// TIA Portal V18 export
VAR_GLOBAL   // PLC tag table "System Variables"
   RotaryCounts AT %MD100 : DInt;   // Actually rotary count feedback
   RotaryRPM AT %MD104 : Real;   // frequency of rotray feedack
   AuxPumpRunning AT %M10.0 : Bool;   // Status of Aux Pump. 1 Running 0 stopped
   EngineRPMCounts AT %MD108 : DInt;   // CAT Engine RPM count return
   EngineRPMFreq AT %MD112 : Real;   // CAT Engine RPM freqency measured
   CoolingFanRunning AT %M10.1 : Bool;   // Status of Cooler Running 0 stopped
   M1Running AT %M10.2 : Bool;   // Status of P1 Running 0 stopped
   M2Running AT %M10.3 : Bool;   // Status of P2 Running 0 stopped
   AuxPumpHOA AT %M10.4 : Bool;   // Actual Signal to Soft Starter
   CoolingFanHOA AT %M10.5 : Bool;   // Actual Signal to Soft Starter
   M1HOA AT %M10.6 : Bool;   // Actual Signal to Soft Starter
   M2HOA AT %M10.7 : Bool;   // Actual Signal to Soft Starter
   ChargePump1PSw AT %M11.0 : Bool;   // Close = Pressure
   TDLubeFlowSw AT %M11.1 : Bool;   // Close = Flow
   TankLowLevelSw AT %M11.2 : Bool;   // Low Level = Open
   TankHighTempSw AT %M11.3 : Bool;   // High Temp = Open
   TDFwdFilter2 AT %M11.5 : Bool;   // Plugged = Open
   TDRevFilter1 AT %M11.6 : Bool;   // Plugged = Open
   TDRevFilter2 AT %M11.7 : Bool;   // Plugged = Open
   AuxReturnFilter AT %M12.0 : Bool;   // Plugged = Open
   KLoopFilter AT %M12.1 : Bool;   // Plugged = Open
   ChargeFilter AT %M12.2 : Bool;   // Plugged = Open
   M1CurrentRaw AT %MW122 : Int;
   M2CurrentRaw AT %MW128 : Int;
   M1CurrentV AT %MD124 : Real;
   M2CurrentV AT %MD130 : Real;
   TDPressFWDRaw AT %MW134 : Int;   // TD Forward Pressure Input
   TDPressREVRaw AT %MW136 : Int;   // TD Reverse Pressure Input
   ClosedLoopTempRaw AT %MW138 : Int;
   ChargeFlowRaw AT %MW140 : Int;
   HotOilShuttleFlowRaw AT %MW142 : Int;
   AuxFlowRaw AT %MW144 : Int;
   ChargePress1Raw AT %MW146 : Int;
   ChargePress2Raw AT %MW148 : Int;
   TDPressFWDmA AT %MD150 : Real;   // TD Forward Pressure Input
   TDPressREVmA AT %MD154 : Real;   // TD Reverse Pressure Input
   ClosedLoopTempmA AT %MD158 : Real;
   ChargeFlowmA AT %MD162 : Real;
   HotOilShuttleFlowmA AT %MD166 : Real;
   AuxFlowmA AT %MD170 : Real;
   ChargePress1mA AT %MD174 : Real;
   ChargePress2mA AT %MD178 : Real;
   TDP1FwdCmdActRaw AT %MW182 : Int;   // Actual measured output to valve from module
   TDP1RevCmdActRaw AT %MW184 : Int;   // Actual measured output to valve from module
   TDP2FwdCmdActRaw AT %MW186 : Int;   // Actual measured output to valve from module
   TDP2RevCmdActRaw AT %MW188 : Int;   // Actual measured output to valve from module
   TDTorqCmdActRaw AT %MW190 : Int;   // Raw Output to card
   TDP1FwdCmdActmA AT %MD192 : Real;   // Actual measured output to valve from module
   TDP1RevCmdActmA AT %MD196 : Real;   // Actual measured output to valve from module
   TDP2FwdCmdActmA AT %MD200 : Real;   // Actual measured output to valve from module
   TDP2RevCmdActmA AT %MD204 : Real;   // Actual measured output to valve from module
   TDTorqCmdActmA AT %MD208 : Real;   // Actual measured output to valve from module
   LinkRetSw AT %M12.4 : Bool;   // Console Input
   TDAuxSw AT %M12.5 : Bool;   // Console Input
   LinkExtSw AT %M12.6 : Bool;   // Console Input
   TDEnSW AT %M12.7 : Bool;   // Console Input
   HSLT_Sw AT %M13.0 : Bool;   // Console Input
   HandlerFwdSw AT %M13.1 : Bool;   // Console Input
   HandlerRevSw AT %M13.2 : Bool;   // Console Input
   MPNotRunning AT %M13.3 : Bool;   // 0 Pump Running, 1 Pump Not Running - Allowed to Run. Power to permit
   QuillLockSw AT %M13.4 : Bool;   // Console Input
   BUWClSw AT %M13.5 : Bool;   // Console Input
   BUWDnSw AT %M13.6 : Bool;   // Console Input
   BUWUpSw AT %M13.7 : Bool;   // Console Input
   TDModeMUSpinSw AT %M14.0 : Bool;   // Console Input
   TDModeMUTorqSw AT %M14.1 : Bool;   // Console Input
   TDModeDrillRevSw AT %M14.2 : Bool;   // Console Input
   TDModeBreakOutSw AT %M14.3 : Bool;   // Console Input
   ElevOpSw AT %M14.4 : Bool;   // Console Input
   TDExtSw AT %M14.5 : Bool;   // Console Input
   ElevClSw AT %M14.6 : Bool;   // Console Input
   TDRetSw AT %M14.7 : Bool;   // Console Input
   PTO_Sw AT %M15.0 : Bool;   // Console Input
   PurgePressureSw AT %M15.1 : Bool;   // Console Input
   MSVClSw AT %M15.2 : Bool;   // Console Input
   MSVAutoSw AT %M15.3 : Bool;   // Console Input
   MSVOpSw AT %M15.4 : Bool;   // Console Input
   LinkFloatSw AT %M15.5 : Bool;   // Console Input
   MUTorqPotRaw AT %MW212 : Int;
   DrillTorqPotRaw AT %MW214 : Int;
   DrillThrottlePotRaw AT %MW216 : Int;
   MUTorqPotV AT %MD218 : Real;
   DrillTorqPotV AT %MD222 : Real;
   DrillThrottlePotV AT %MD226 : Real;
   RotEncLDSlot AT %MB230 : Byte;   // Bit 0-3 Slot 0, Bit 4-7 Slot 1. 0 0 0 0 for Idle, 0 0 0 1 Load Counter
   TDFwdPress1Raw AT %MD240 : UDInt;   // Pump 1 Forward Pressure output
   TDFwdPress2Raw AT %MD244 : UDInt;   // Pump 2 Forward Pressure output
   TDRevPress1Raw AT %MD248 : UDInt;   // Pump 1 Rev Pressure output
   TDRevPress2Raw AT %MD252 : UDInt;   // Pump 2 Rev Pressure output
   TDTorqPressRaw AT %MD256 : UDInt;   // Torq Output
   TDFwdPress1En AT %M15.6 : Bool;   // Enable Pump 1 Forward Pressure output
   TDFwdPress2En AT %M15.7 : Bool;   // Enable Pump 2 Forward Pressure output
   TDRevPress1En AT %M16.0 : Bool;   // Enable Pump 1 Rev Pressure output
   TDRevPress2En AT %M16.1 : Bool;   // Enable Pump 2 Rev Pressure output
   TDTorqPressEn AT %M16.2 : Bool;   // Enable Torq output
   BUWClSol AT %M16.4 : Bool;
   HSLT_Sol AT %M16.5 : Bool;
   ElevClSol AT %M16.6 : Bool;
   ElevOpSol AT %M16.7 : Bool;
   LinkExtSol AT %M17.0 : Bool;
   LinkRetSol AT %M17.1 : Bool;
   LinkFloatSol AT %M17.2 : Bool;
   LSHT_Sol AT %M17.3 : Bool;
   MSVOpSol AT %M17.4 : Bool;
   MSVClSol AT %M17.5 : Bool;
   BUWDnSol AT %M17.6 : Bool;
   BUWUpSol AT %M17.7 : Bool;
   HandlerFWDSol AT %M18.0 : Bool;
   HandlerREVSol AT %M18.1 : Bool;
   TDExtSol AT %M18.2 : Bool;
   TDRetSol AT %M18.3 : Bool;   // Output Coil
   HourMeterOn AT %M18.4 : Bool;
   EngRampSpeedDn AT %M18.5 : Bool;
   AuxPumpStart AT %M18.6 : Bool;
   EngRampSpeedUp AT %M18.7 : Bool;
   CoolingFanStart AT %M19.0 : Bool;
   FailSafeEnSol AT %M19.1 : Bool;
   PumpEnSol AT %M19.2 : Bool;   // CAT/Rig 11 Only
   BOControlSol AT %M19.3 : Bool;
   AuxUnloaderSol AT %M19.4 : Bool;
   HotOilControlSol AT %M19.5 : Bool;
   BUWOpSol AT %M19.6 : Bool;
   BypassValveSol AT %M19.7 : Bool;
   TDFwdPress1mA AT %MD260 : Real;   // Pump 1 Forward Pressure output
   TDFwdPress2mA AT %MD264 : Real;   // Pump 2 Forward Pressure output
   TDRevPress1mA AT %MD268 : Real;   // Pump 1 Rev Pressure output
   TDRevPress2mA AT %MD272 : Real;   // Pump 2 Rev Pressure output
   TDTorqPressmA AT %MD276 : Real;   // Torq Output
   PTOLED AT %M20.4 : Bool;
   HPUFaultLED AT %M20.5 : Bool;
   TDFlushFaultLED AT %M20.6 : Bool;
   BUWClLED AT %M20.7 : Bool;
   TDEnLED AT %M21.0 : Bool;
   ConLowPurgeLED AT %M21.1 : Bool;
   MSVClLED AT %M21.2 : Bool;   // Mud Saver valve closed LED
   QuillLockLED AT %M21.3 : Bool;
   ElevClLED AT %M21.4 : Bool;
   Horn AT %M21.5 : Bool;
   MSVClInt AT %M21.6 : Bool;   // Mud saver valve closed interlocks outputs
   BUWClInt AT %M21.7 : Bool;   // BUW Closed interlock outputs
   DrillRecTorqRaw AT %MW280 : Int;
   DrillRecRPMRaw AT %MW282 : Int;
   DrillRecTorqFtLbs AT %MD284 : Real;
   DrillRecRPM AT %MD288 : Real;
   DrillRecTorqmA AT %MD292 : Real;
   DrillRecRPMmA AT %MD296 : Real;
   RotEncUnFl AT %M22.0 : Bool;   // Encoder underflow
   RotEncOvFl AT %M22.1 : Bool;   // Encoder OVerflow
   RotEncPosReset AT %M22.2 : Bool;   // Set high to trigger zero position of encoder. Bit will reset once position reset
   RotEncSlot0 AT %MD232 : Real;
   RotEncSlot1 AT %MD236 : Real;
   TDRotStopped AT %M22.3 : Bool;   // Set if TD has not moved after stop time elapsed
   RotAbsPosDeg AT %MD300 : Real;   // Absolute rotary position from zero point
   RotRelPosDeg AT %MD304 : Real;   // Position from 0-360 degrees
   RotPosTurns AT %MD308 : Real;   // Turns from zero point
   TDFlushFlowSw AT %M22.4 : Bool;
   M1Current AT %MD312 : Real;
   M2Current AT %MD316 : Real;
   TDPressFwdPSI AT %MD320 : Real;   // TD Fwd Pressure PSI
   TDPressRevPSI AT %MD324 : Real;   // TD Rev Pressure PSI
   ClosedLoopTempC AT %MD328 : Real;   // Closed Loop Temp in C
   ChargeFlowGPM AT %MD332 : Real;   // Charge Flow in GPM
   HotOilFlowGPM AT %MD336 : Real;   // Hot Oil Shuttle Flow in GPM
   AuxFlowGPM AT %MD340 : Real;   // Aux Flow GPM
   ChargePress1PSI AT %MD344 : Real;   // Charge Pump 1 Pressure PSI
   ChargePress2PSI AT %MD348 : Real;   // Charge Pump 2 Pressure PSI
   M1CurrentFilt AT %MD352 : Real;
   M2CurrentFilt AT %MD356 : Real;
   TDPressFwdPSIFilt AT %MD360 : Real;
   TDPressRevPSIFilt AT %MD364 : Real;
   ClosedLoopTempCFilt AT %MD368 : Real;
   ChargeFlowGPMFilt AT %MD372 : Real;
   HotOilFlowGPMFilt AT %MD376 : Real;
   AuxFlowGPMFilt AT %MD380 : Real;
   ChargePress1PSIFilt AT %MD384 : Real;
   ChargePress2PSIFilt AT %MD388 : Real;
   AuxPumpHand AT %M22.5 : Bool;   // Starter HOA switch in the Hand Position
   AuxPumpOff AT %M22.6 : Bool;   // Starter HOA switch in the Off position
   CoolingFanHand AT %M23.0 : Bool;   // Starter HOA switch in the Hand Position
   CoolingFanOff AT %M23.1 : Bool;   // Starter HOA switch in the Off position
   M1Hand AT %M23.3 : Bool;   // Starter HOA switch in the Hand Position
   M1Off AT %M23.4 : Bool;   // Starter HOA switch in the Off position
   M2Hand AT %M23.6 : Bool;   // Starter HOA switch in the Hand Position
   M2Off AT %M23.7 : Bool;   // Starter HOA switch in the Off position
   AuxPumpFault AT %M22.7 : Bool;   // Motor failed to start before motor timeout time
   CoolingFanFault AT %M23.2 : Bool;   // Motor failed to start before motor timeout time
   M1Fault AT %M23.5 : Bool;   // Motor failed to start before motor timeout time
   M2Fault AT %M24.0 : Bool;   // Motor failed to start before motor timeout time
   M1Start AT %M20.2 : Bool;   // Start Motor 1
   M2Start AT %M20.3 : Bool;   // Start Motor 2
   BypassStart AT %M24.1 : Bool;   // Ready for Bypass to start, waiting for PTO
   BypassRunning AT %M24.2 : Bool;   // Latched Signal set if PTO pressed after Bypass Start
   StartCAT AT %M24.3 : Bool;   // Indicates CAT startup up. System ramps up and will enable.
   BUWMaintConfirm AT %M24.4 : Bool;
   PTOConfirmed AT %M24.5 : Bool;   // PTO Confirm pulse for 5 seconds after button pressed
   BUWOpenClk AT %M24.6 : Bool;   // Periodic clock signal that will be on for 5 seconds and off for 1 min. Used for maintain gripper open
   BUWAutoCl AT %M24.7 : Bool;   // Latch for Gripper Close
   BUWAutoClHold AT %M25.0 : Bool;   // LAtch for Gripper Hold Closed
   BUWAutoOp AT %M25.1 : Bool;   // Lath for Gripper Open
   OscSpeedfwdHold AT %M25.2 : Bool;
   QuillLockEnabled AT %M25.3 : Bool;   // Bit used to know if Quill Lock allowed
   BUWClHoldTime AT %M25.4 : Bool;   // On for half a second to hold the close before turning off
   MUTorqPotPer AT %MD392 : Real;
   DrillTorqPotPer AT %MD396 : Real;
   DrillThrottlePotPer AT %MD400 : Real;
   MUTorqPotPerFilt AT %MD404 : Real;
   DrillTorqPotPerFilt AT %MD408 : Real;
   DrillThrottlePotPerFilt AT %MD412 : Real;
   ActTorqFtLbs AT %MD416 : Real;   // Calculated actual torque
   ActTorqFtLbsFilt AT %MD420 : Real;   // Filtered Actual Torque
   TDDifPressPSI AT %MD424 : Real;   // Diffential pressure betweeen FWD and REV
   DrillTorqSetFtLbs AT %MD428 : Real;   // Internal setpoint value from the console input FtLbs
   MUTorqSetFtLbs AT %MD432 : Real;   // Internal setpoint value from the console input FtLbs
   RotDegPerCount AT %MD436 : Real;   // Actual Degrees per Count for current encoder setup
   DrillTorqSetMax AT %MD440 : Real;   // Maximum value allowed to set drill torq too based on MU torq settings
   BOCycleDone AT %M25.6 : Bool;   // Trigger when BO Sw released
   MUCycleDone AT %M25.7 : Bool;   // Set when MU done
   MUSwRelease AT %M26.0 : Bool;   // Trigger when MU SW released
   MUDoneSetFtLbs AT %MD444 : Real;   // Minimum torque to surpass to declare MU Done
   ElevClFeedback AT %M12.3 : Bool;   // Feedback switch that the elevators are closed
   LamptTest AT %M26.1 : Bool;   // Bit Used to trigger Lamp to turn on.
   FlushFaultNoSpin AT %M26.2 : Bool;   // TD flush faulted. No Spin allowed
   ThrottleDisable AT %M26.3 : Bool;   // Throttle disable if high
   ThrottleUnlocked AT %M26.4 : Bool;   // Throttle boots up locked. Must be below zero to enable after startup
   DrillTorqLimited AT %M26.5 : Bool;   // Set high if max drill torq limited by max makeup torq
   DrillTorqSetPSI AT %MD448 : Real;   // PSI equivalent to get desired torq from valve
   MUTorqSetPSI AT %MD452 : Real;   // PSI equivalent to get desired torq from valve
   TDStart AT %M25.5 : Bool;   // Bit will be set High when TD is started for regular operations
   BypassPTO AT %M26.6 : Bool;   // Bypass PTO accept
   BypassOutEnable AT %M26.7 : Bool;   // Bypass control enabled to allow signal to Pumps after delay
   BypassHighTemp AT %M27.0 : Bool;   // High Closed loop temp in bypass mode
   TDPressTxFault AT %M27.1 : Bool;   // One of the pressure transducers if not working. No auto MU
   HSLTDisThrottle AT %M27.2 : Bool;   // Bit high after shift to disable throttle
   LSHTDisThrottle AT %M27.3 : Bool;   // Bit high after shift to disable throttle
   MUSeqRunning AT %M27.4 : Bool;   // Bool indicating mak up sequence is running.
   AutoMUTorqLow AT %M27.5 : Bool;   // Auto Make Up Low Torque range
   AutoMUTorqMid AT %M27.6 : Bool;   // Auto Make Up Mid Torque Range
   AutoMuTorqHigh AT %M27.7 : Bool;   // Auto Make Up High Torque Range
   HiTempRPMRed AT %M28.1 : Bool;   // Bit indicating high temperature and RPM to be reduced
   HiTempShutdown AT %M28.2 : Bool;   // Bit indicating high temperature and shutdown needed.
   TDRotDirFwd AT %M28.3 : Bool;   // Rotary moving fwd
   TDRotDirRev AT %M28.4 : Bool;   // Rotary moving rev
   ActTorqKFtLbsFilt AT %MD456 : Real;
   RotEncA AT %M28.5 : Bool;
   RotEncB AT %M28.6 : Bool;
   BOSeqRunning AT %M28.0 : Bool;   // Bool indicating break out sequence is running.   {ExternalVisible false}
   HPU_AiV2SpareRaw AT %MW460 : Int;   // Spare Analog Voltage Input Raw
   HPU_AiV2SpareV AT %MD472 : Real;   // Spare Analog Voltage Input
   HPU_AiV3SpareRaw AT %MW462 : Int;   // Spare Analog Voltage Input Raw
   HPU_AiV4SpareRaw AT %MW464 : Int;   // Spare Analog Voltage Input Raw
   HPU_AiV5SpareRaw AT %MW466 : Int;   // Spare Analog Voltage Input Raw
   HPU_AiV6SpareRaw AT %MW468 : Int;   // Spare Analog Voltage Input Raw
   HPU_AiV7SpareRaw AT %MW470 : Int;   // Spare Analog Voltage Input Raw
   HPU_AiV3SpareV AT %MD476 : Real;   // Spare Analog Voltage Input
   HPU_AiV4SpareV AT %MD480 : Real;   // Spare Analog Voltage Input
   HPU_AiV5SpareV AT %MD484 : Real;   // Spare Analog Voltage Input
   HPU_AiV6SpareV AT %MD488 : Real;   // Spare Analog Voltage Input
   HPU_AiV7SpareV AT %MD492 : Real;   // Spare Analog Voltage Input
   Con_AiV3SpareRaw AT %MW496 : Int;   // Spare Analog Voltage Input Raw
   Con_AiV4SpareRaw AT %MW498 : Int;   // Spare Analog Voltage Input Raw
   Con_AiV5SpareRaw AT %MW500 : Int;   // Spare Analog Voltage Input Raw
   Con_AiV6SpareRaw AT %MW502 : Int;   // Spare Analog Voltage Input Raw
   Con_AiV7SpareRaw AT %MW504 : Int;   // Spare Analog Voltage Input Raw
   Con_AiV3SpareV AT %MD506 : Real;   // Spare Analog Voltage Input
   Con_AiV4SpareV AT %MD510 : Real;   // Spare Analog Voltage Input
   Con_AiV5SpareV AT %MD514 : Real;   // Spare Analog Voltage Input
   Con_AiV6SpareV AT %MD518 : Real;   // Spare Analog Voltage Input
   Con_AiV7SpareV AT %MD522 : Real;   // Spare Analog Voltage Input
   HornTest AT %M28.7 : Bool;
   Charge1Fault AT %M29.0 : Bool;   // Charge pressure fault while TD enabled
   FilterPlugged AT %M29.1 : Bool;
   Clock_Byte AT %MB0 : Byte;
   Clock_10Hz AT %M0.0 : Bool;   // 0.1 s period
   Clock_5Hz AT %M0.1 : Bool;   // 0.2 s period
   "Clock_2.5Hz" AT %M0.2 : Bool;   // 0.4 s period
   Clock_2Hz AT %M0.3 : Bool;   // .06 s period
   "Clock_1.25Hz" AT %M0.4 : Bool;   // 0.8s period
   Clock_1Hz AT %M0.5 : Bool;   // 1s period
   "Clock_0.625Hz" AT %M0.6 : Bool;   // 1.6s period
   "Clock_0.5Hz" AT %M0.7 : Bool;   // 2.0 s period
   HiTempAlarm AT %M29.2 : Bool;
   LubeFlowFault AT %M29.3 : Bool;
   HornSilence AT %M29.4 : Bool;
   EngineFault AT %M29.5 : Bool;   // CAT Engine Fault. Below min RPM
   EngineRPM AT %MD116 : Real;
   ClosedLoopTempCMax AT %MD526 : Real;
   TDEnabled AT %M16.3 : Bool;   // Start Request received and system enabled
   Charge2Fault AT %M20.0 : Bool;
   ChargePump2PSw AT %M29.7 : Bool;   // Close = Pressure
   TDFwdFilter1 AT %M11.4 : Bool;   // Plugged = Open
   LastCount AT %MD30 : DInt;
   RotRelPosDegHMIPos AT %MD34 : Real;
   OscHomeRelDegHMIPos AT %MD530 : Real;
   SwitchSWGATE AT %M538.0 : Bool;
   OscSpeedrevHold AT %M38.0 : Bool;
   RevFwdPause AT %M38.1 : Bool;
   FwdRevPasue AT %M38.2 : Bool;
   PSIadjustbit AT %M38.3 : Bool;
   PSIdrillTorquCalca AT %MD540 : Real;
   PSIsettle AT %MD548 : Real;
   PSIadjustRange AT %MD552 : Real;
   PSIadjustval AT %MD556 : Real;
   ClosedLoopTempF AT %MD560 : Real;
   RotaryRPMActual AT %MD564 : Real;
END_VAR
VAR_GLOBAL CONSTANT   // user constants
   AlwaysOn : Bool := 1;
   AlwaysOff : Bool := 0;
END_VAR
